// TIA Portal V19 export
DATA_BLOCK "ControlNodes"   // DB94
// stored: MemoryReserve 100, Namespace Unit2.EM0
   VAR
      em { ExternalWritable := 'False'} : "LAF_typeEmControlNode";
      jobs { ExternalWritable := 'False'} : "LAF_typeJobs";
      sequence { ExternalWritable := 'False'} : "LAF_typeSequence";
   END_VAR
BEGIN
   em.status.enabled := true;
END_DATA_BLOCK
